FUNCTION_BLOCK FB_GantryDiffVirtualLimitSwitch
VAR_INPUT
	PEnc	:	ST_RenishawEnc;
	SEnc	:	ST_RenishawEnc;
	
	GantDiffTol	:	LINT;
END_VAR
VAR_OUTPUT
	PLimFwd		:	BOOL;
	PLimBwd		:	BOOL;
	
	SLimFwd		:	BOOL;
	SLimBwd		:	BOOL;
END_VAR
VAR
	GantryDiff	:	LINT;
END_VAR

(* Gantry Difference Virtual Limit Switch
A. Wallace 17-2-15

Determines which direction is disabled due to it increasing the gantry difference.
Refer to the ESD for actual conventions.

A positive gantry error refers to a CCW clocked assembly:
eg. for X
X1 upstream, X2 downstream. Primary axis is always upstream.
Gantry difference > 0 when
X2>X1
Therefore
X2 positive direction disabled
X1 negative direction disabled

Call before FB_MotionStage fb calls for the gantry axes.
*)

GantryDiff := ( ULINT_TO_LINT(PEnc.Count) - ULINT_TO_LINT(PEnc.Ref) ) - ( ULINT_TO_LINT(SEnc.Count) - ULINT_TO_LINT(SEnc.Ref) );

IF ABS(GantryDiff) > GantDiffTol THEN
	IF GantryDiff < 0  THEN
		PLimBwd := FALSE;
		SLimFwd := FALSE;
	ELSE	
		PLimBwd := TRUE;
		SLimFwd := TRUE;
	END_IF
	IF GantryDiff > 0 THEN
		PLimFwd := FALSE;
		SLimBwd := FALSE;
	ELSE
		PLimFwd := TRUE;
		SLimBwd := TRUE;
	END_IF
ELSE
	//If there is no fault, all directions are enabled
	PLimFwd := TRUE;
	PLimBwd := TRUE;
	SLimFwd := TRUE;
	SLimBwd := TRUE;
END_IF

END_FUNCTION_BLOCK

(* stored: Version 1.1.0.1, ProductVersion 3.1.4022.18
   POU FB_GantryDiffVirtualLimitSwitch: Id {ae668e37-4b4c-400f-bda9-27f8d308d0b6}, SpecialFunc None *)
